FUNCTION_BLOCK AE2_SPLIT_MERGE (* Bidirectional Splitter and Merger, no Forwarding between SOCKET and PLUG *)
  (* Standard: 61499-2; Function: Any Event coming in by SOCKET or PLUG is output at EO, Any Event from EI is splitted to SOCKET and PLUG; Description: Copyright (c) 2025 HR Agrartechnik GmbH This program and the accompanying materials are made available under the terms of the Eclipse Public License 2.0 which is available at https://www.eclipse.org/legal/epl-2.0/ SPDX-License-Identifier: EPL-2.0 *)
  (* Version 1.0, 2025-01-24, Franz Höpfinger, HR Agrartechnik GmbH *)
  PACKAGE adapter::events::bidirectional;
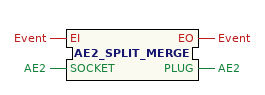
  EVENT_INPUT
    EI; (* Input Event *)
  END_EVENT
  EVENT_OUTPUT
    EO; (* Output Event *)
  END_EVENT
  SOCKETS
    SOCKET : adapter::types::bidirectional::AE2;
  END_SOCKETS
  PLUGS
    PLUG : adapter::types::bidirectional::AE2;
  END_PLUGS
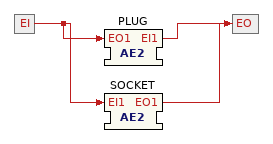
  EVENT_CONNECTIONS
    PLUG.EI1 TO EO;
    SOCKET.EO1 TO EO;
    EI TO PLUG.EO1;
    EI TO SOCKET.EI1;
  END_CONNECTIONS
END_FUNCTION_BLOCK
